{attribute 'qualified_only'}
{attribute 'strict'}
{attribute 'to_string'}
TYPE DUT_Command_ArrayType :
(
	StoredPosition := 0,
	VisionRegister := 1,
	Flag := 2
);
END_TYPE

(* stored: Version 1.1.0.1
   EnumerationTextList DUT_Command_ArrayType: Id {17560b0c-5c79-43ac-95f8-43d98381b6d0} *)
